// TIA Portal project "scl_3buton_2motor_kontrol" (V18)

(* hardware
DEVICE "S7-1200 station_1"  S7-1200 Station
   slot 0: "Rack_0"  S7-1200 Rack  Rack  V1.0
   slot 1: "PLC_1"  CPU 1214C DC/DC/DC  6ES7 214-1AG40-0XB0  V4.6
*)

// ===== PLC "PLC_1"  CPU 1214C DC/DC/DC =====

VAR_GLOBAL   // PLC tag table "Default tag table"
   "STOP" AT %I0.0 : Bool;
   "START_1" AT %I0.1 : Bool;
   "START_2" AT %I0.2 : Bool;
   "MOTOR_1" AT %Q0.0 : Bool;
   "MOTOR_2" AT %Q0.1 : Bool;
END_VAR

FUNCTION "Block_1" : Void   // FC1, SCL
{ S7_Optimized_Access := 'TRUE' }
VERSION : 0.1
BEGIN
   IF "START_1"=1 THEN

       "MOTOR_1" := 1;

   END_IF;
   IF "START_2" = 1 AND "START_1" = 1 THEN
       "MOTOR_1" := 0;
       "MOTOR_2" := 1;

   END_IF;
   IF "STOP"=1 THEN
       "MOTOR_1" := 0;
       "MOTOR_2" := 0;
   END_IF;
END_FUNCTION

ORGANIZATION_BLOCK "Main"   // OB1, LAD, ProgramCycle
TITLE = "Main Program Sweep (Cycle)"
{ S7_Optimized_Access := 'TRUE' }
VERSION : 0.1
// UYGULAMA-3: 3 buton ile 2 pikis kontrol edilecektir.
// *1. Buton ile 1. Çikis sürekli çalisir.
// 2. Buton ile 1. Çikis durur, 2. Çikis sürekli çalisir.
// Buton ile 1. Çikis ve 2. Gikis durur.
   VAR_INPUT
      Initial_Call : Bool;   // Initial call of this OB
      Remanence : Bool;   // =True, if remanent data are available
   END_VAR
BEGIN
END_ORGANIZATION_BLOCK